Fanuc KAREL source: ka00090.KL

-- PROVISIONAL review KL for V940-1; original PC SHA256 b703a6681be139e4e8253f2da784e5ab78a8f2cc436f21cb757f8a9004bc22f0
-- Incomplete behavior may be omitted. Consult companion uncertainty JSON. Do not deploy.
PROGRAM KA00090
%NOLOCKGROUP
-- UNRESOLVED_DECL SRC type=000199
-- UNRESOLVED_DECL DST type=000102
BEGIN
  -- V9_ZERO_TABLE_METADATA_HINT layout=0001; no indexed target words; source/name/runtime held
  -- UNRESOLVED_PC offsets 5-25; opcodes 49,7E,4A
  -- UNRESOLVED_PC offsets 30-34; opcodes 7F
END KA00090
